// TIA Portal V19 export
FUNCTION_BLOCK "Network XC208"   // FB10, LAD
{ S7_Optimized_Access := 'TRUE' }
// stored: MemoryReserve 100, SetENOAutomatically false
   VAR_INPUT
      Trigger : Bool;   // Trigger the network scan for port info, rising edge
      HWID : HW_ANY;   // Scalance Interface of the switch
   END_VAR
   VAR_OUTPUT
      Error : Bool;
      Status : Word;
   END_VAR
   VAR_IN_OUT
      NetworkHMI_PortInfo : Variant;   // HMI input and output interface
   END_VAR
   VAR
      PortInformation { S7_SetPoint := 'True'} : "LPNDR_ReadGlobalInfo";   // LPNDR mode returns Port Information
   END_VAR
   VAR CONSTANT
      modeInterfaceInformation : Int := 1;
      modeMRPInformation : Int := 2;
      modePortInformation : Int := 3;
      modePortLinkStatus : Int := 4;
      modePortStatistics : Int := 5;
   END_VAR
BEGIN

REGION Network 1: Mode 3: Read Port Information
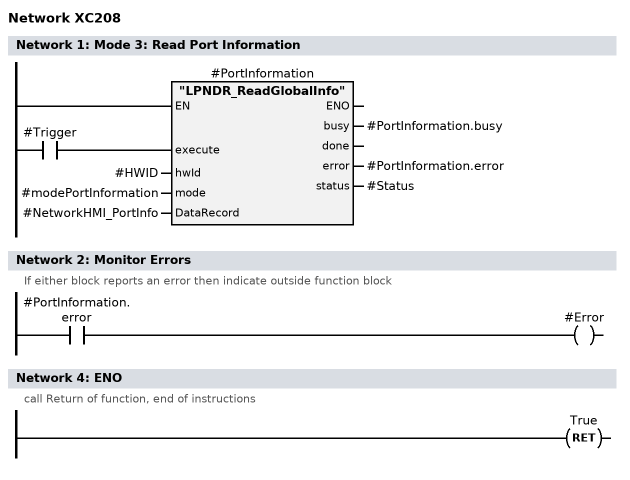
   RUNG wire#powerrail
      #PortInformation(execute := wire#w1, hwId := #HWID, mode := #modePortInformation, DataRecord := #NetworkHMI_PortInfo, busy => #PortInformation.busy, done =>, error => #PortInformation.error, status => #Status)
   END_RUNG
   RUNG wire#powerrail
      Contact( #Trigger )
   END_RUNG wire#w1
   // the same network as SCL:
   #PortInformation(execute := #Trigger,   // "LPNDR_ReadGlobalInfo"
                    hwId := #HWID,
                    mode := #modePortInformation,
                    DataRecord := #NetworkHMI_PortInfo,
                    busy => #PortInformation.busy,
                    error => #PortInformation.error,
                    status => #Status);
END_REGION

REGION Network 2: Monitor Errors
   // If either block reports an error then indicate outside function block
   RUNG wire#powerrail
      Contact( #PortInformation.error )
      Coil( #Error )
   END_RUNG
   // the same network as SCL:
   #Error := #PortInformation.error;
END_REGION

REGION Network 3
   // #Port."Port" := #Port.Ports[#Index];
END_REGION

REGION Network 4: ENO
   // call Return of function, end of instructions
   ENO := True;
   RETURN;
END_REGION
END_FUNCTION_BLOCK
